FUNCTION_BLOCK ConveyorSC
VAR_INPUT
	bEnable : BOOL;
END_VAR
VAR_OUTPUT
	trueMode : ConveyorMode;
	requestedMode : ConveyorMode;
	
	error AT %I* : BOOL;
	position AT %I* : REAL;
	velocity AT %I* : REAL;
END_VAR
VAR
	enable AT %Q* : BOOL := TRUE;
	direction AT %Q* : BOOL; //FALSE = forward, TRUE = backward
	pulse AT %Q* : BOOL;
	reset AT %Q* : BOOL;
	
	sensorEntry AT %I* : BOOL := TRUE;
	sensorExit AT %I* : BOOL;
END_VAR
VAR
	//nextConveyor : POINTER TO ConveyorSC;
	//prevConveyor : POINTER TO ConveyorSC;
	
	pulser : TP; //pulses are assumed to be low-high-low
END_VAR
VAR_STAT CONSTANT
	pulseWidth : TIME := T#50MS;
END_VAR

enable := bEnable;

override();

sequence();

METHOD backward : BOOL
VAR_INPUT
END_VAR
END_METHOD

METHOD forward : BOOL
VAR_INPUT
END_VAR
END_METHOD

{attribute 'monitoring' := 'call'}
PROPERTY IsOccupied : BOOL
GET
IsOccupied := sensorExit OR sensorEntry;
END_GET
END_PROPERTY

METHOD join : BOOL
VAR_INPUT
	conveyor : POINTER TO ConveyorSC;
END_VAR
//nextConveyor := conveyor;
//conveyor^.prevConveyor := THIS;
END_METHOD

METHOD PROTECTED override : BOOL
VAR_INPUT
END_VAR
END_METHOD

METHOD reset : BOOL
VAR_INPUT
END_VAR
position := 0;
velocity := velocity; //no change
END_METHOD

METHOD PROTECTED sequence : BOOL
VAR_INPUT
END_VAR
direction := (trueMode = ConveyorMode.BACKWARD); //set direction bit

pulser(IN:= , PT:= pulseWidth, Q=> pulse, ET=> );
pulser.IN := 
	enable AND 
	NOT error AND 
	NOT reset AND 
	(trueMode = ConveyorMode.FORWARD OR trueMode = ConveyorMode.BACKWARD)
	AND pulser.Q; //ends pulse itself
END_METHOD

METHOD setMode : BOOL
VAR_INPUT
	mode : ConveyorMode;
END_VAR
trueMode := mode;
END_METHOD

METHOD setRequest : BOOL
VAR_INPUT
	newRequest : ConveyorMode;
END_VAR
requestedMode := newRequest;
END_METHOD

METHOD target : BOOL
VAR_INPUT
	targetPosition : REAL;
END_VAR
END_METHOD

END_FUNCTION_BLOCK

(* stored: Version 1.1.0.1, ProductVersion 3.1.4024.11
   POU ConveyorSC: Id {d3063b85-1d0e-4601-ab41-5fdef5457493}, SpecialFunc None
   Folder Private: Id {1a888f12-4db7-4903-9f4c-6c8f1d797dc1}
   Folder Properties: Id {1765f27b-9fb2-425e-b273-a472c5a609e9}
   Folder Unused: Id {1c2f1e14-da9a-4098-b511-317af27de399}
   Method backward: Id {e8202226-4ec6-4684-856e-619a6d551d16}
   Method forward: Id {1da2a125-0c3e-4b60-939d-889602df2c25}
   Property IsOccupied: Id {b0b7aab6-d707-4fd5-b282-0025795c566b}
   Get Get: Id {cf0344a5-3161-4da7-ba48-678c5bd761bd}
   Method join: Id {a0cf54f0-e20b-4bf6-a83b-b1805adbdb65}
   Method override: Id {8e6f4597-0bc4-436a-ab2a-8db6201b5164}
   Method reset: Id {bc427059-4ffe-412e-a00d-70dfddb646fc}
   Method sequence: Id {4423a6bc-d34b-4c46-82c9-1d91c2591f42}
   Method setMode: Id {5dc00876-44a2-4178-b0ed-3fd9c716e599}
   Method setRequest: Id {87bf1b84-a271-46b8-9a30-1c3e8e6aad73}
   Method target: Id {cbc2aa81-2d60-42f2-80e1-cf506a3bd543} *)
